INTERFACE IStation

PROPERTY Position : REFERENCE TO FB_Position
GET
END_GET
SET
END_SET
END_PROPERTY

PROPERTY Process : REFERENCE TO FB_AUT_ABSTRACT
GET
END_GET
SET
END_SET
END_PROPERTY

END_INTERFACE

(* stored: Version 1.1.0.1, ProductVersion 3.1.4024.6
   Itf IStation: Id {fa1d6360-5f8e-4b4c-8b1d-5d83c2a9962d}
   Property Position: Id {42fce230-3fd5-4649-9ed7-60495560311f}
   Get Get: Id {651463c6-131b-4577-99ae-702213c4c5e2}
   Set Set: Id {f2c2670a-ec9b-4eda-9a0b-32a350131516}
   Property Process: Id {01bf1ff3-01ac-4306-934d-936c8f13119a}
   Get Get: Id {65b5f7fc-d95f-44a2-a294-f1e92ddb1ed5}
   Set Set: Id {3f6c809e-81de-404b-831f-a0485c893482} *)
